(* IEC 61131-3 sources: PLC_02/ArCan/ArCanSend, 3 files *)

(* ---- Action.st ---- *)
ACTION ActionArCanSender:

	CASE ArCanSender.step OF
		STEP_WAIT:
			(* wait for starting *)
			IF (ArCanSender.enable = TRUE) THEN
				ArCanSender.step := STEP_INIT_BAUDRATE;
			END_IF;

		STEP_INIT_BAUDRATE: (* Initializes the sender with ArCanSetBaudrate to 250 kbit/s *)
			ArCanSender.ArCanSetBaudrate_0.Execute := TRUE;
			ArCanSender.ArCanSetBaudrate_0.DeviceName := ArCanSender.senderDeviceName;
			ArCanSender.ArCanSetBaudrate_0.Baudrate := ArCanSender.Baudrate;		(* Set to 250 000 bit/s *)

			ArCanSender.ArCanSetBaudrate_0();

			IF (ArCanSender.ArCanSetBaudrate_0.Done = TRUE) THEN
				gSignalCheck.Can_HardwareCheck2 := TRUE;
				ArCanSender.step := STEP_INIT_SENDER;
			ELSIF (ArCanSender.ArCanSetBaudrate_0.Error = TRUE) THEN
				ArCanSender.lastError := ArCanSender.ArCanSetBaudrate_0.StatusID;
				ArCanSender.errorCount := ArCanSender.errorCount + 1;
				ArCanSender.step := STEP_ERROR;
			END_IF;

		STEP_INIT_SENDER:	(* Initializes the CAN Sender *)
			ArCanSender.ArCanSend_0.Enable := TRUE;
			ArCanSender.ArCanSend_0.DeviceName := ArCanSender.senderDeviceName;

			IF (ArCanSender.ArCanSend_0.Active = TRUE) THEN		(* Checks if the FB is active for configuring a sending CAN frame *)
				ArCanSender.step := STEP_WAIT_CMD;
				gSignalCheck.Can_SendCheck := TRUE;
			ELSIF (ArCanSender.ArCanSend_0.Error = TRUE) THEN
				ArCanSender.errorCount := ArCanSender.errorCount + 1;
				ArCanSender.lastError := ArCanSender.ArCanSend_0.StatusID;
				ArCanSender.step := STEP_ERROR;
			END_IF;

		STEP_WAIT_CMD:

			IF (ArCanSender.enable = FALSE) THEN (* User stops the test *)
				ArCanSender.step := STEP_DEINIT;
			END_IF;

		STEP_INIT_SEND_FRAME: (* Transmits a CAN Frame *)

			IF (ArCanSender.ArCanSend_0.NumberOfFreeBuffers > 0) THEN

				ArCanSender.ArCanSend_0.Frame.DataLength := 8;
				ArCanSender.ArCanSend_0.Frame.ID := ArCanSender.ID;
				ArCanSender.ArCanSend_0.Frame.Format := ArCanSender.Format;
				ArCanSender.ArCanSend_0.SendFrame := TRUE;	(* Copies the frame into the internal buffer for sending it *)

				ArCanSender.successCount := ArCanSender.successCount + 1;	(* Frame is in the queue and will be sent *)
			ELSE
				ArCanSender.ArCanSend_0.SendFrame := FALSE;
				ArCanSender.waitCounter := ArCanSender.waitCounter  + 1; (* Interface has no more free internal buffers *)
			END_IF;

			IF (ArCanSender.ArCanSend_0.Error = TRUE) THEN
				ArCanSender.lastError := ArCanSender.ArCanSend_0.StatusID;
				ArCanSender.errorCount := ArCanSender.errorCount + 1;
				ArCanSender.step := STEP_ERROR;
			END_IF;

			IF (ArCanSender.enable = FALSE) THEN (* User stops the test *)
				ArCanSender.step := STEP_DEINIT;
			END_IF;

		STEP_DEINIT:
			ArCanSender.ArCanSend_0.Enable := FALSE;
			ArCanSender.step := STEP_WAIT;

		STEP_ERROR:
			ArCanSender.ArCanSend_0.Enable := FALSE;
			IF (ArCanSender.enable = FALSE) THEN (* User stops the test *)
				ArCanSender.step := STEP_DEINIT;
			END_IF;

	END_CASE;

	ArCanSender.ArCanSend_0();

END_ACTION

(* ---- ArCanSend.st ---- *)
// CAN_CH_A

PROGRAM _INIT

	ArCanSender.enable				:= TRUE;

	(* CAN parameter configuration *)
	ArCanSender.senderDeviceName 	:= 'IF7';       (* for X20CP0482 CPU *)
//	ArCanSender.senderDeviceName 	:= 'IF1.ST2.IF1.ST2.IF1';		(* for C50 Touch Panel + X20CS2770 *)
	ArCanSender.Baudrate			:= 125000;		(* Set to 500 000 bit/s *)

	ArCanSender.Format				:= arCAN_29BIT; // or arCAN_29BIT

	(**********	 CAN Baud rate Baudrate Value	************)
	(*******************************************************)
	(* 	  1 000 000 bit/s    >>		Baudrate = 1000000	   *)
	(* 		800 000 bit/s    >>		Baudrate =  800000	   *)
	(* 		500 000 bit/s    >>		Baudrate =  500000	   *)
	(* 		250 000 bit/s    >>		Baudrate =  250000	   *)
	(* 		125 000 bit/s    >>		Baudrate =  125000	   *)
	(* 		100 000 bit/s    >>		Baudrate =  100000	   *)
	(* 		050 000 bit/s    >>		Baudrate =  50000	   *)
	(* 		020 000 bit/s    >>		Baudrate =  20000	   *)
	(* 		010 000 bit/s    >>		Baudrate =  10000	   *)
	(*******************************************************)
	(*******************************************************)

END_PROGRAM

PROGRAM _CYCLIC

	timerCount				:= timerCount + 1;
	IF timerCount >= 2 THEN     // ( cycle time x 5 ) = time for step change (2ms x 5 = 10ms)
		timerCount	:= 0;
		step				:= step + 1;
		IF step > 9 THEN        // after the last step 9, go back to 0 step
			step	:= 0;
		END_IF
		IF ArCanSender.step = STEP_WAIT_CMD THEN
			ArCanSender.step	:= STEP_INIT_SEND_FRAME;
		END_IF
	END_IF

	(***********************************************************)
	(* Customize the sending data *)

	CASE step OF
		0:
			ArCanSender.ID							:= 16#06080000;
			ArCanSender.ArCanSend_0.Frame.Data[0]	:= CharMD0.TxFunCode;
			ArCanSender.ArCanSend_0.Frame.Data[1]	:= 0;
			ArCanSender.ArCanSend_0.Frame.Data[2]	:= UINT_TO_BYTE(SHR(CharMD0.TxRegNum, 8));
			ArCanSender.ArCanSend_0.Frame.Data[3]	:= UINT_TO_BYTE(CharMD0.TxRegNum AND 16#FF );
			ArCanSender.ArCanSend_0.Frame.Data[4]	:= UDINT_TO_BYTE(SHR(CharMD0.TxData_Set, 24));
			ArCanSender.ArCanSend_0.Frame.Data[5]	:= UDINT_TO_BYTE(SHR(CharMD0.TxData_Set, 16));
			ArCanSender.ArCanSend_0.Frame.Data[6]	:= UDINT_TO_BYTE(SHR(CharMD0.TxData_Set, 8));
		    ArCanSender.ArCanSend_0.Frame.Data[7]	:= UDINT_TO_BYTE(CharMD0.TxData_Set AND 16#000000FF);

		1:
			ArCanSender.ID							:= 16#06080800;
			ArCanSender.ArCanSend_0.Frame.Data[0]	:= CharMD1.TxFunCode;
			ArCanSender.ArCanSend_0.Frame.Data[1]	:= 0;
			ArCanSender.ArCanSend_0.Frame.Data[2]	:= UINT_TO_BYTE(SHR(CharMD1.TxRegNum, 8));
			ArCanSender.ArCanSend_0.Frame.Data[3]	:= UINT_TO_BYTE	(CharMD1.TxRegNum AND 16#FF );
			ArCanSender.ArCanSend_0.Frame.Data[4]	:= UDINT_TO_BYTE(SHR(CharMD1.TxData_Set, 24));
			ArCanSender.ArCanSend_0.Frame.Data[5]	:= UDINT_TO_BYTE(SHR(CharMD1.TxData_Set, 16));
			ArCanSender.ArCanSend_0.Frame.Data[6]	:= UDINT_TO_BYTE(SHR(CharMD1.TxData_Set, 8));
			ArCanSender.ArCanSend_0.Frame.Data[7]	:= UDINT_TO_BYTE(CharMD1.TxData_Set AND 16#000000FF);

	END_CASE

	(***********************************************************)

	IF (ArCanSender.successCount <> successCountOld) THEN
		successCountOld						:= ArCanSender.successCount;
		ArCanSender.ArCanSend_0.SendFrame	:= FALSE;
		ArCanSender.step					:= STEP_WAIT_CMD;
	END_IF

	(* Action for Sender *)
	ActionArCanSender;

END_PROGRAM

PROGRAM _EXIT
	(* Deinitialization of the sender *)
	ArCanSender.ArCanSend_0.Enable := FALSE;
	ArCanSender.ArCanSend_0();
END_PROGRAM

(* ---- ArCanSend.var ---- *)
VAR
	ArCanSender : ArCanSend_typ;
	step : USINT;
	successCountOld : UDINT;
	timerCount : UDINT;
END_VAR
